TEXTLIST equivalenciaBaldaOcupada
  TRUE = 'Ocupada'
  FALSE = 'Libre'
   = ''
END_TEXTLIST

(* stored: Version 1.1.0.1, ProductVersion 3.1.4024.15
   TextList equivalenciaBaldaOcupada: Id {4eacc289-8466-4bd2-bac8-bf8962b6df9f} *)
